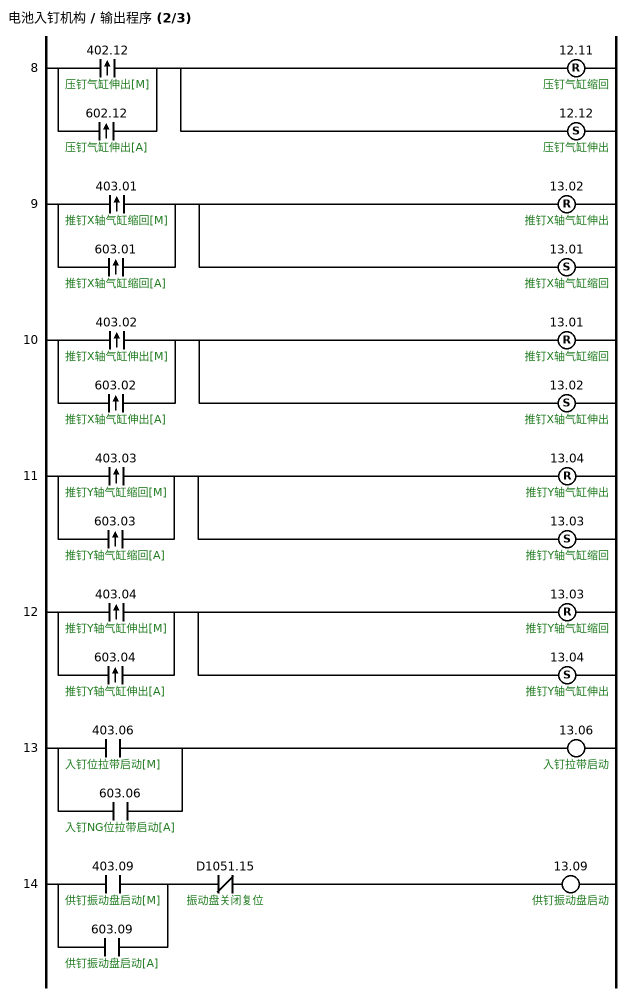
; [picture p120: 电池入钉机构 / 输出程序, rungs 8-14]
; rung 8
@LD 402.12  ; 压钉气缸伸出[M]
@OR 602.12  ; 压钉气缸伸出[A]
RSET 12.11  ; 压钉气缸缩回
SET 12.12  ; 压钉气缸伸出
; rung 9
@LD 403.01  ; 推钉X轴气缸缩回[M]
@OR 603.01  ; 推钉X轴气缸缩回[A]
RSET 13.02  ; 推钉X轴气缸伸出
SET 13.01  ; 推钉X轴气缸缩回
; rung 10
@LD 403.02  ; 推钉X轴气缸伸出[M]
@OR 603.02  ; 推钉X轴气缸伸出[A]
RSET 13.01  ; 推钉X轴气缸缩回
SET 13.02  ; 推钉X轴气缸伸出
; rung 11
@LD 403.03  ; 推钉Y轴气缸缩回[M]
@OR 603.03  ; 推钉Y轴气缸缩回[A]
RSET 13.04  ; 推钉Y轴气缸伸出
SET 13.03  ; 推钉Y轴气缸缩回
; rung 12
@LD 403.04  ; 推钉Y轴气缸伸出[M]
@OR 603.04  ; 推钉Y轴气缸伸出[A]
RSET 13.03  ; 推钉Y轴气缸缩回
SET 13.04  ; 推钉Y轴气缸伸出
; rung 13
LD 403.06  ; 入钉位拉带启动[M]
OR 603.06  ; 入钉NG位拉带启动[A]
OUT 13.06  ; 入钉拉带启动
; rung 14
LD 403.09  ; 供钉振动盘启动[M]
OR 603.09  ; 供钉振动盘启动[A]
ANDNOT D1051.15  ; 振动盘关闭复位
OUT 13.09  ; 供钉振动盘启动

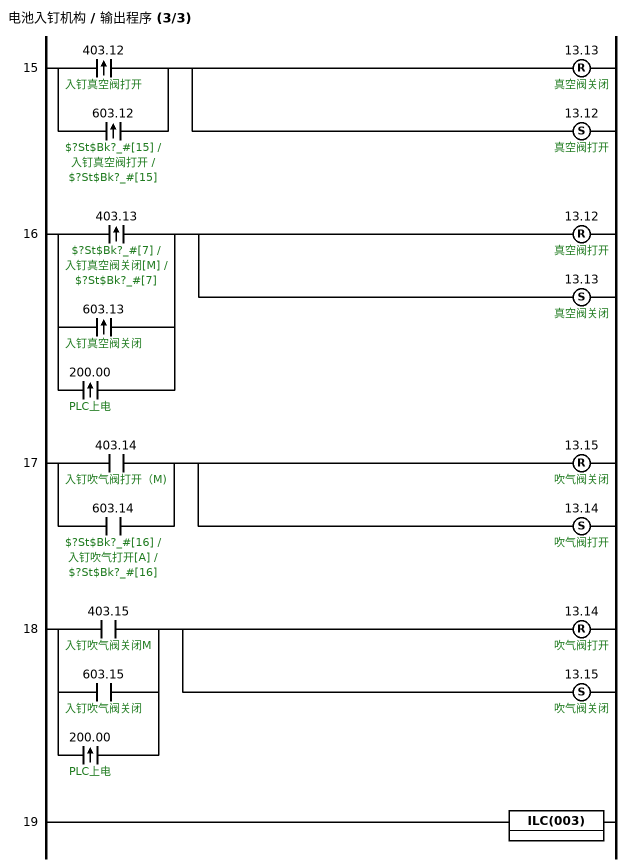
; rung 15
@LD 403.12  ; 入钉真空阀打开
@OR 603.12  ; $?St$Bk?_#[15] / 入钉真空阀打开 / $?St$Bk?_#[15]
RSET 13.13  ; 真空阀关闭
SET 13.12  ; 真空阀打开
; rung 16
@LD 403.13  ; $?St$Bk?_#[7] / 入钉真空阀关闭[M] / $?St$Bk?_#[7]
@OR 603.13  ; 入钉真空阀关闭
@OR 200.00  ; PLC上电
RSET 13.12  ; 真空阀打开
SET 13.13  ; 真空阀关闭
; rung 17
LD 403.14  ; 入钉吹气阀打开（M)
OR 603.14  ; $?St$Bk?_#[16] / 入钉吹气打开[A] / $?St$Bk?_#[16]
RSET 13.15  ; 吹气阀关闭
SET 13.14  ; 吹气阀打开
; rung 18
LD 403.15  ; 入钉吹气阀关闭M
OR 603.15  ; 入钉吹气阀关闭
@OR 200.00  ; PLC上电
RSET 13.14  ; 吹气阀打开
SET 13.15  ; 吹气阀关闭
; rung 19
ILC(003)

### Section 入钉升降伺服参数

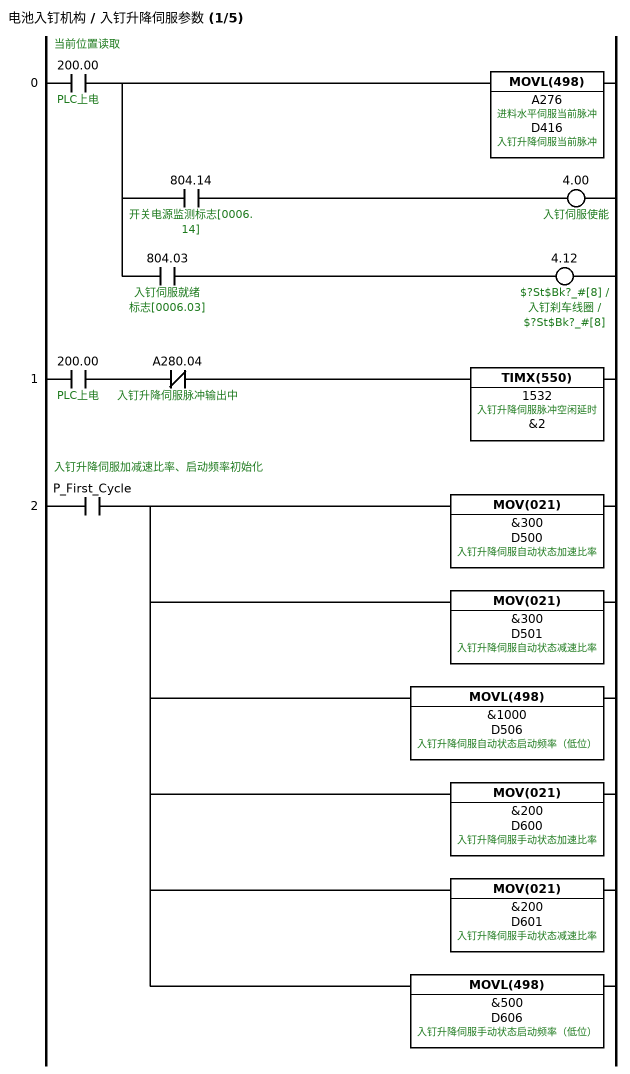
; rung 0: 当前位置读取
LD 200.00  ; PLC上电
OUT TR0
MOVL(498) A276 D416  ; 进料水平伺服当前脉冲, 入钉升降伺服当前脉冲
AND 804.14  ; 开关电源监测标志[0006.14]
OUT 4.00  ; 入钉伺服使能
LD TR0
AND 804.03  ; 入钉伺服就绪 标志[0006.03]
OUT 4.12  ; $?St$Bk?_#[8] / 入钉刹车线圈 / $?St$Bk?_#[8]
; rung 1
LD 200.00  ; PLC上电
ANDNOT A280.04  ; 入钉升降伺服脉冲输出中
TIMX(550) 1532 &2  ; 入钉升降伺服脉冲空闲延时
; rung 2: 入钉升降伺服加减速比率、启动频率初始化
LD P_First_Cycle
MOV(021) &300 D500  ; 入钉升降伺服自动状态加速比率
MOV(021) &300 D501  ; 入钉升降伺服自动状态减速比率
MOVL(498) &1000 D506  ; 入钉升降伺服自动状态启动频率（低位）
MOV(021) &200 D600  ; 入钉升降伺服手动状态加速比率
MOV(021) &200 D601  ; 入钉升降伺服手动状态减速比率
MOVL(498) &500 D606  ; 入钉升降伺服手动状态启动频率（低位）

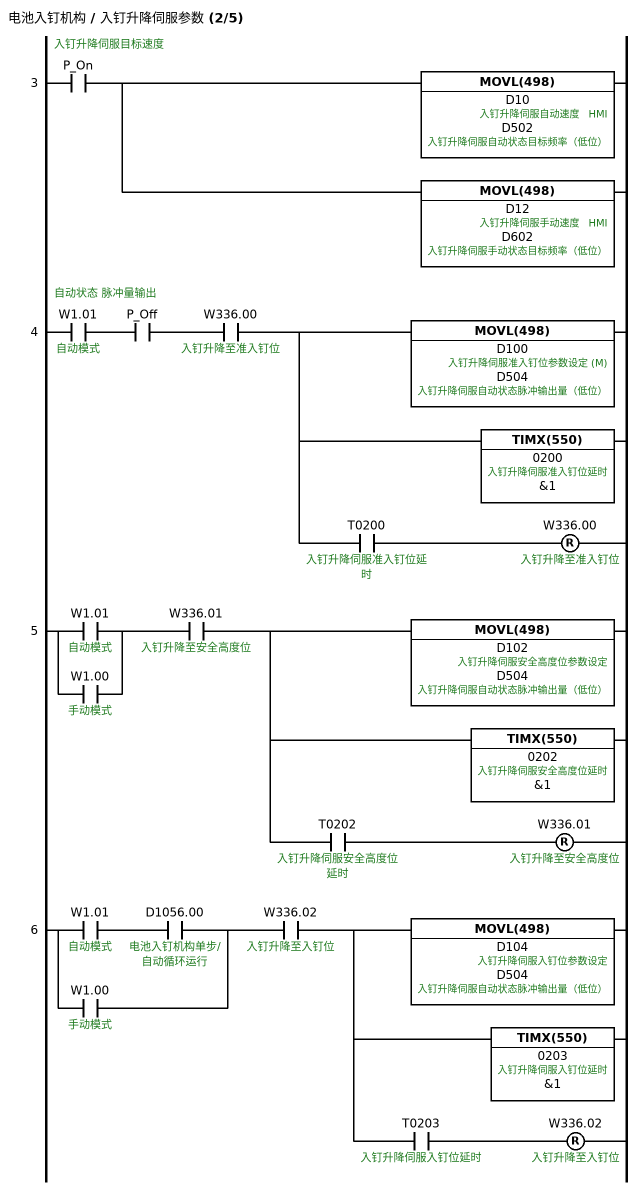
; rung 3: 入钉升降伺服目标速度
LD P_On
MOVL(498) D10 D502  ; 入钉升降伺服自动速度   HMI, 入钉升降伺服自动状态目标频率（低位）
MOVL(498) D12 D602  ; 入钉升降伺服手动速度   HMI, 入钉升降伺服手动状态目标频率（低位）
; rung 4: 自动状态 脉冲量输出
LD W1.01  ; 自动模式
AND P_Off
AND W336.00  ; 入钉升降至准入钉位
MOVL(498) D100 D504  ; 入钉升降伺服准入钉位参数设定 (M), 入钉升降伺服自动状态脉冲输出量（低位）
TIMX(550) 0200 &1  ; 入钉升降伺服准入钉位延时
AND T0200  ; 入钉升降伺服准入钉位延时
RSET W336.00  ; 入钉升降至准入钉位
; rung 5
LD W1.01  ; 自动模式
OR W1.00  ; 手动模式
AND W336.01  ; 入钉升降至安全高度位
MOVL(498) D102 D504  ; 入钉升降伺服安全高度位参数设定, 入钉升降伺服自动状态脉冲输出量（低位）
TIMX(550) 0202 &1  ; 入钉升降伺服安全高度位延时
AND T0202  ; 入钉升降伺服安全高度位延时
RSET W336.01  ; 入钉升降至安全高度位
; rung 6
LD W1.01  ; 自动模式
AND D1056.00  ; 电池入钉机构单步/自动循环运行
OR W1.00  ; 手动模式
AND W336.02  ; 入钉升降至入钉位
MOVL(498) D104 D504  ; 入钉升降伺服入钉位参数设定, 入钉升降伺服自动状态脉冲输出量（低位）
TIMX(550) 0203 &1  ; 入钉升降伺服入钉位延时
AND T0203  ; 入钉升降伺服入钉位延时
RSET W336.02  ; 入钉升降至入钉位

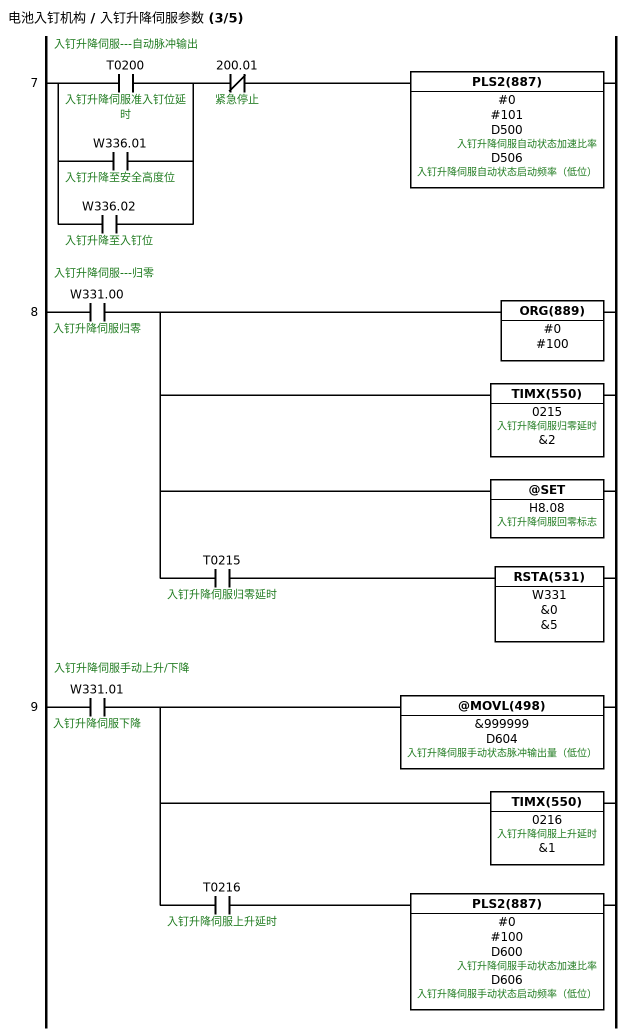
; rung 7: 入钉升降伺服---自动脉冲输出
LD T0200  ; 入钉升降伺服准入钉位延时
OR W336.01  ; 入钉升降至安全高度位
OR W336.02  ; 入钉升降至入钉位
ANDNOT 200.01  ; 紧急停止
PLS2(887) #0 #101 D500 D506  ; 入钉升降伺服自动状态加速比率, 入钉升降伺服自动状态启动频率（低位）
; rung 8: 入钉升降伺服---归零
LD W331.00  ; 入钉升降伺服归零
ORG(889) #0 #100
TIMX(550) 0215 &2  ; 入钉升降伺服归零延时
@SET H8.08  ; 入钉升降伺服回零标志
AND T0215  ; 入钉升降伺服归零延时
RSTA(531) W331 &0 &5
; rung 9: 入钉升降伺服手动上升/下降
LD W331.01  ; 入钉升降伺服下降
@MOVL(498) &999999 D604  ; 入钉升降伺服手动状态脉冲输出量（低位）
TIMX(550) 0216 &1  ; 入钉升降伺服上升延时
AND T0216  ; 入钉升降伺服上升延时
PLS2(887) #0 #100 D600 D606  ; 入钉升降伺服手动状态加速比率, 入钉升降伺服手动状态启动频率（低位）

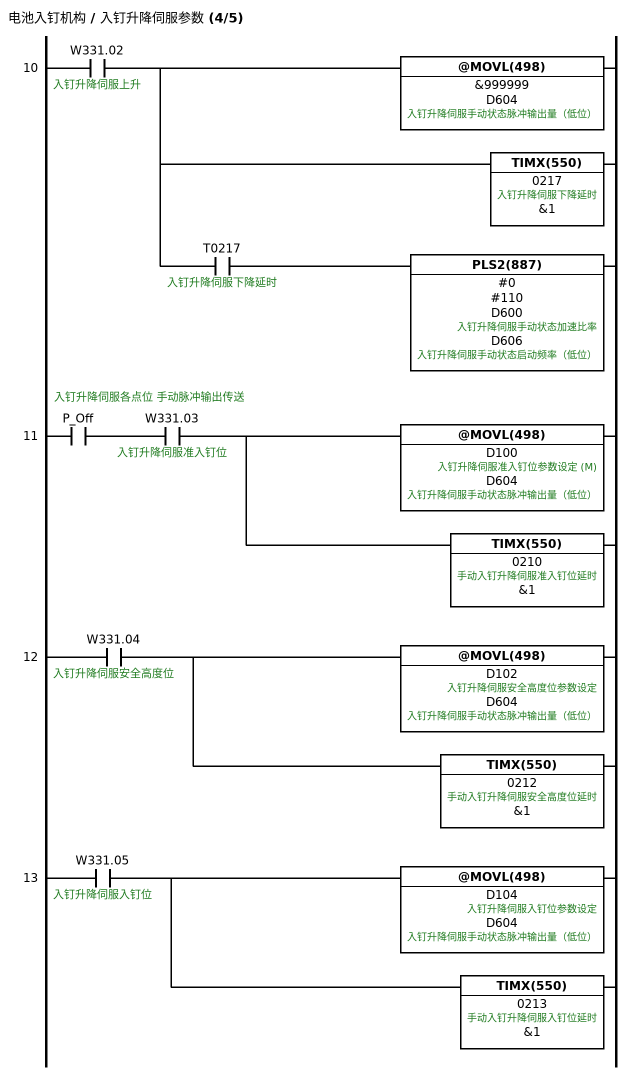
; rung 10
LD W331.02  ; 入钉升降伺服上升
@MOVL(498) &999999 D604  ; 入钉升降伺服手动状态脉冲输出量（低位）
TIMX(550) 0217 &1  ; 入钉升降伺服下降延时
AND T0217  ; 入钉升降伺服下降延时
PLS2(887) #0 #110 D600 D606  ; 入钉升降伺服手动状态加速比率, 入钉升降伺服手动状态启动频率（低位）
; rung 11: 入钉升降伺服各点位 手动脉冲输出传送
LD P_Off
AND W331.03  ; 入钉升降伺服准入钉位
@MOVL(498) D100 D604  ; 入钉升降伺服准入钉位参数设定 (M), 入钉升降伺服手动状态脉冲输出量（低位）
TIMX(550) 0210 &1  ; 手动入钉升降伺服准入钉位延时
; rung 12
LD W331.04  ; 入钉升降伺服安全高度位
@MOVL(498) D102 D604  ; 入钉升降伺服安全高度位参数设定, 入钉升降伺服手动状态脉冲输出量（低位）
TIMX(550) 0212 &1  ; 手动入钉升降伺服安全高度位延时
; rung 13
LD W331.05  ; 入钉升降伺服入钉位
@MOVL(498) D104 D604  ; 入钉升降伺服入钉位参数设定, 入钉升降伺服手动状态脉冲输出量（低位）
TIMX(550) 0213 &1  ; 手动入钉升降伺服入钉位延时

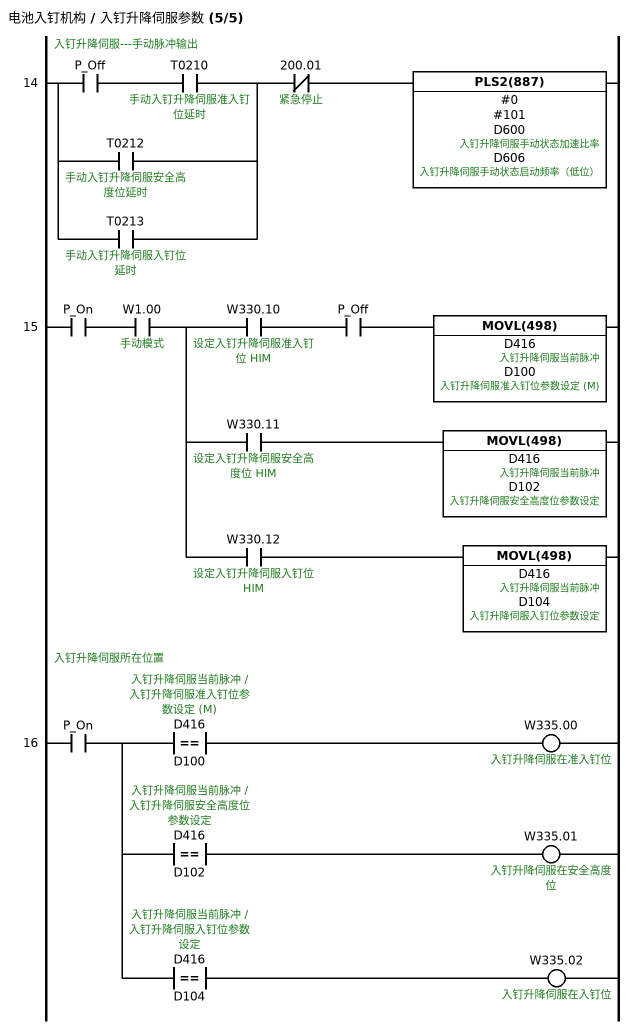
; rung 14: 入钉升降伺服---手动脉冲输出
LD P_Off
AND T0210  ; 手动入钉升降伺服准入钉位延时
OR T0212  ; 手动入钉升降伺服安全高度位延时
OR T0213  ; 手动入钉升降伺服入钉位延时
ANDNOT 200.01  ; 紧急停止
PLS2(887) #0 #101 D600 D606  ; 入钉升降伺服手动状态加速比率, 入钉升降伺服手动状态启动频率（低位）
; rung 15
LD P_On
AND W1.00  ; 手动模式
OUT TR0
AND W330.10  ; 设定入钉升降伺服准入钉位 HIM
AND P_Off
MOVL(498) D416 D100  ; 入钉升降伺服当前脉冲, 入钉升降伺服准入钉位参数设定 (M)
LD TR0
AND W330.11  ; 设定入钉升降伺服安全高度位 HIM
MOVL(498) D416 D102  ; 入钉升降伺服当前脉冲, 入钉升降伺服安全高度位参数设定
LD TR0
AND W330.12  ; 设定入钉升降伺服入钉位 HIM
MOVL(498) D416 D104  ; 入钉升降伺服当前脉冲, 入钉升降伺服入钉位参数设定
; rung 16: 入钉升降伺服所在位置
LD P_On
OUT TR0
AND=SL(303) D416 D100  ; 入钉升降伺服当前脉冲, 入钉升降伺服准入钉位参数设定 (M)
OUT W335.00  ; 入钉升降伺服在准入钉位
LD TR0
AND=SL(303) D416 D102  ; 入钉升降伺服当前脉冲, 入钉升降伺服安全高度位参数设定
OUT W335.01  ; 入钉升降伺服在安全高度位
LD TR0
AND=SL(303) D416 D104  ; 入钉升降伺服当前脉冲, 入钉升降伺服入钉位参数设定
OUT W335.02  ; 入钉升降伺服在入钉位

### Section 入钉旋转步进参数

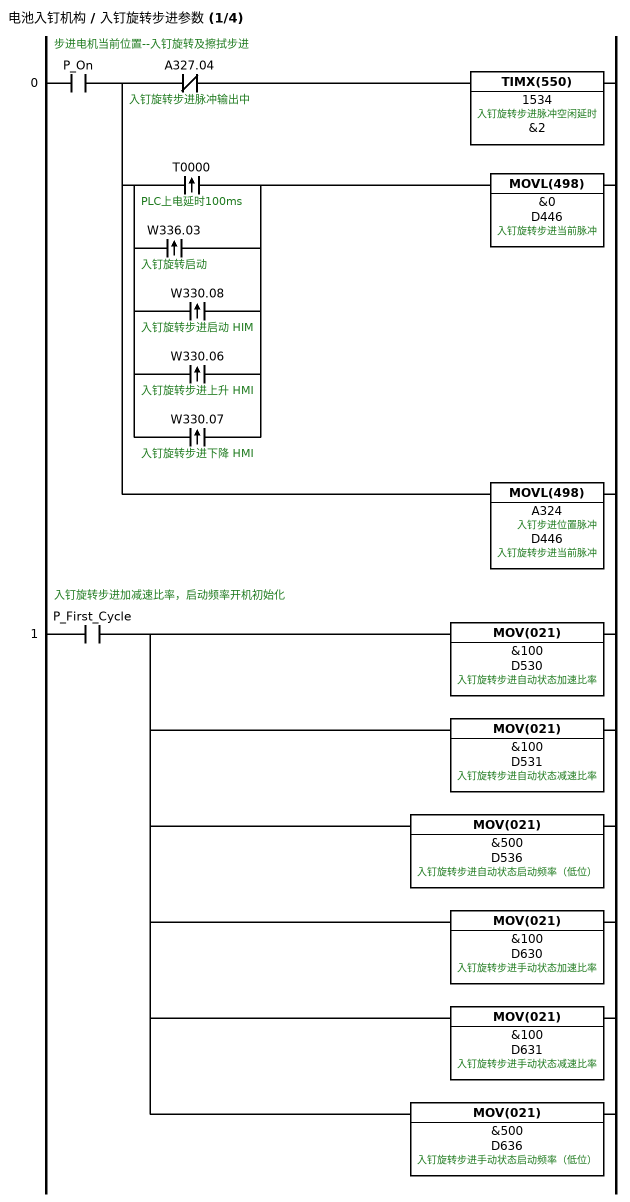
; rung 0: 步进电机当前位置--入钉旋转及擦拭步进
LD P_On
OUT TR0
ANDNOT A327.04  ; 入钉旋转步进脉冲输出中
TIMX(550) 1534 &2  ; 入钉旋转步进脉冲空闲延时
LD TR0
@LD T0000  ; PLC上电延时100ms
@OR W336.03  ; 入钉旋转启动
@OR W330.08  ; 入钉旋转步进启动 HIM
@OR W330.06  ; 入钉旋转步进上升 HMI
@OR W330.07  ; 入钉旋转步进下降 HMI
ANDLD
MOVL(498) &0 D446  ; 入钉旋转步进当前脉冲
LD TR0
MOVL(498) A324 D446  ; 入钉步进位置脉冲, 入钉旋转步进当前脉冲
; rung 1: 入钉旋转步进加减速比率，启动频率开机初始化
LD P_First_Cycle
MOV(021) &100 D530  ; 入钉旋转步进自动状态加速比率
MOV(021) &100 D531  ; 入钉旋转步进自动状态减速比率
MOV(021) &500 D536  ; 入钉旋转步进自动状态启动频率（低位）
MOV(021) &100 D630  ; 入钉旋转步进手动状态加速比率
MOV(021) &100 D631  ; 入钉旋转步进手动状态减速比率
MOV(021) &500 D636  ; 入钉旋转步进手动状态启动频率（低位）

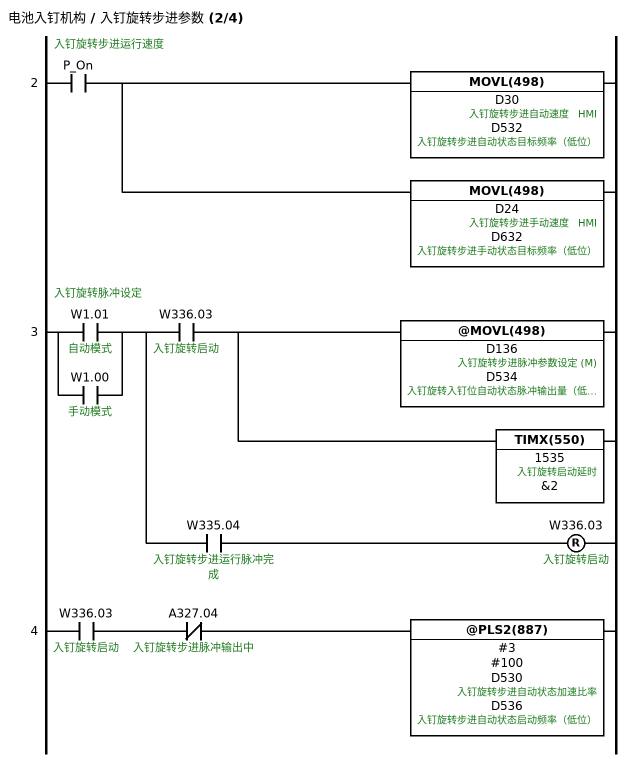
; rung 2: 入钉旋转步进运行速度
LD P_On
MOVL(498) D30 D532  ; 入钉旋转步进自动速度   HMI, 入钉旋转步进自动状态目标频率（低位）
MOVL(498) D24 D632  ; 入钉旋转步进手动速度   HMI, 入钉旋转步进手动状态目标频率（低位）
; rung 3: 入钉旋转脉冲设定
LD W1.01  ; 自动模式
OR W1.00  ; 手动模式
OUT TR0
AND W336.03  ; 入钉旋转启动
@MOVL(498) D136 D534  ; 入钉旋转步进脉冲参数设定 (M), 入钉旋转入钉位自动状态脉冲输出量（低位）
TIMX(550) 1535 &2  ; 入钉旋转启动延时
LD TR0
AND W335.04  ; 入钉旋转步进运行脉冲完成
RSET W336.03  ; 入钉旋转启动
; rung 4
LD W336.03  ; 入钉旋转启动
ANDNOT A327.04  ; 入钉旋转步进脉冲输出中
@PLS2(887) #3 #100 D530 D536  ; 入钉旋转步进自动状态加速比率, 入钉旋转步进自动状态启动频率（低位）

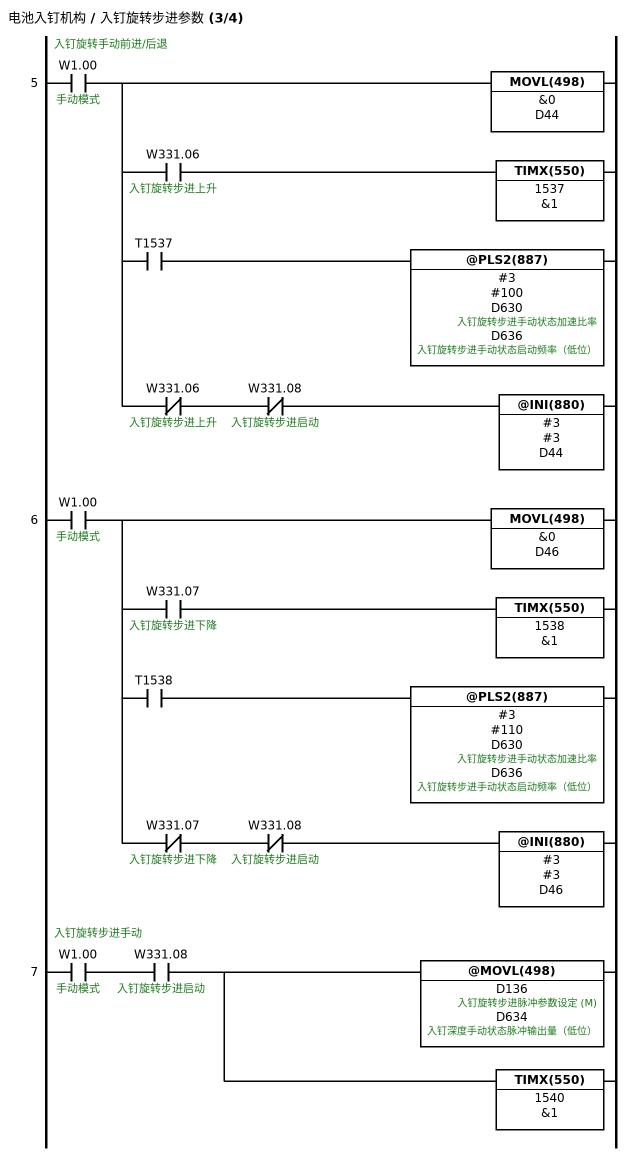
; rung 5: 入钉旋转手动前进/后退
LD W1.00  ; 手动模式
OUT TR0
MOVL(498) &0 D44
AND W331.06  ; 入钉旋转步进上升
TIMX(550) 1537 &1
LD TR0
AND T1537
@PLS2(887) #3 #100 D630 D636  ; 入钉旋转步进手动状态加速比率, 入钉旋转步进手动状态启动频率（低位）
LD TR0
ANDNOT W331.06  ; 入钉旋转步进上升
ANDNOT W331.08  ; 入钉旋转步进启动
@INI(880) #3 #3 D44
; rung 6
LD W1.00  ; 手动模式
OUT TR0
MOVL(498) &0 D46
AND W331.07  ; 入钉旋转步进下降
TIMX(550) 1538 &1
LD TR0
AND T1538
@PLS2(887) #3 #110 D630 D636  ; 入钉旋转步进手动状态加速比率, 入钉旋转步进手动状态启动频率（低位）
LD TR0
ANDNOT W331.07  ; 入钉旋转步进下降
ANDNOT W331.08  ; 入钉旋转步进启动
@INI(880) #3 #3 D46
; rung 7: 入钉旋转步进手动
LD W1.00  ; 手动模式
AND W331.08  ; 入钉旋转步进启动
@MOVL(498) D136 D634  ; 入钉旋转步进脉冲参数设定 (M), 入钉深度手动状态脉冲输出量（低位）
TIMX(550) 1540 &1

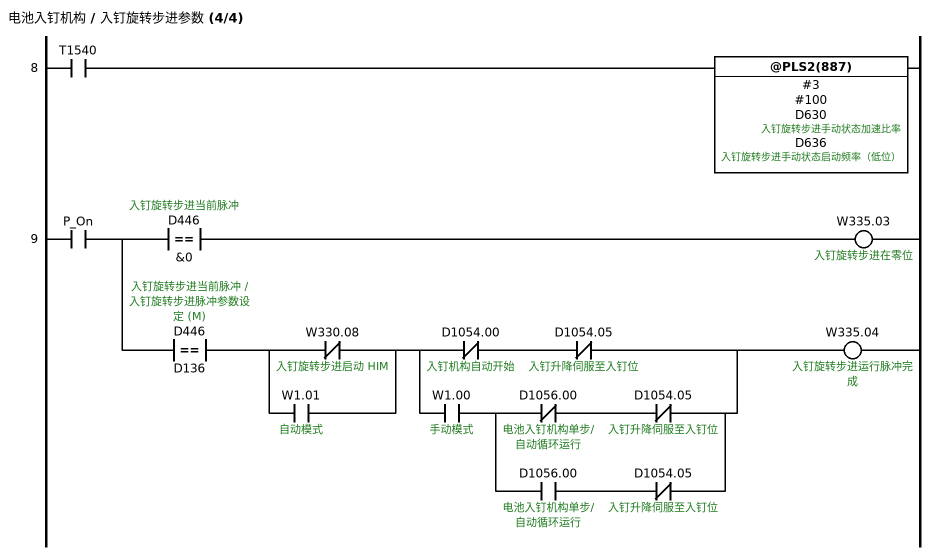
; rung 8
LD T1540
@PLS2(887) #3 #100 D630 D636  ; 入钉旋转步进手动状态加速比率, 入钉旋转步进手动状态启动频率（低位）
; rung 9
LD P_On
OUT TR0
AND=SL(303) D446 &0  ; 入钉旋转步进当前脉冲
OUT W335.03  ; 入钉旋转步进在零位
LD TR0
AND=SL(303) D446 D136  ; 入钉旋转步进当前脉冲, 入钉旋转步进脉冲参数设定 (M)
LDNOT W330.08  ; 入钉旋转步进启动 HIM
OR W1.01  ; 自动模式
ANDLD
LDNOT D1054.00  ; 入钉机构自动开始
ANDNOT D1054.05  ; 入钉升降伺服至入钉位
LD W1.00  ; 手动模式
LDNOT D1056.00  ; 电池入钉机构单步/自动循环运行
ANDNOT D1054.05  ; 入钉升降伺服至入钉位
LD D1056.00  ; 电池入钉机构单步/自动循环运行
ANDNOT D1054.05  ; 入钉升降伺服至入钉位
ORLD
ANDLD
ORLD
ANDLD
OUT W335.04  ; 入钉旋转步进运行脉冲完成

### Section END
; rung 0
END(001)

## Program 入钉NG抓取机构 (cyclic task 5)

### Section 主程序

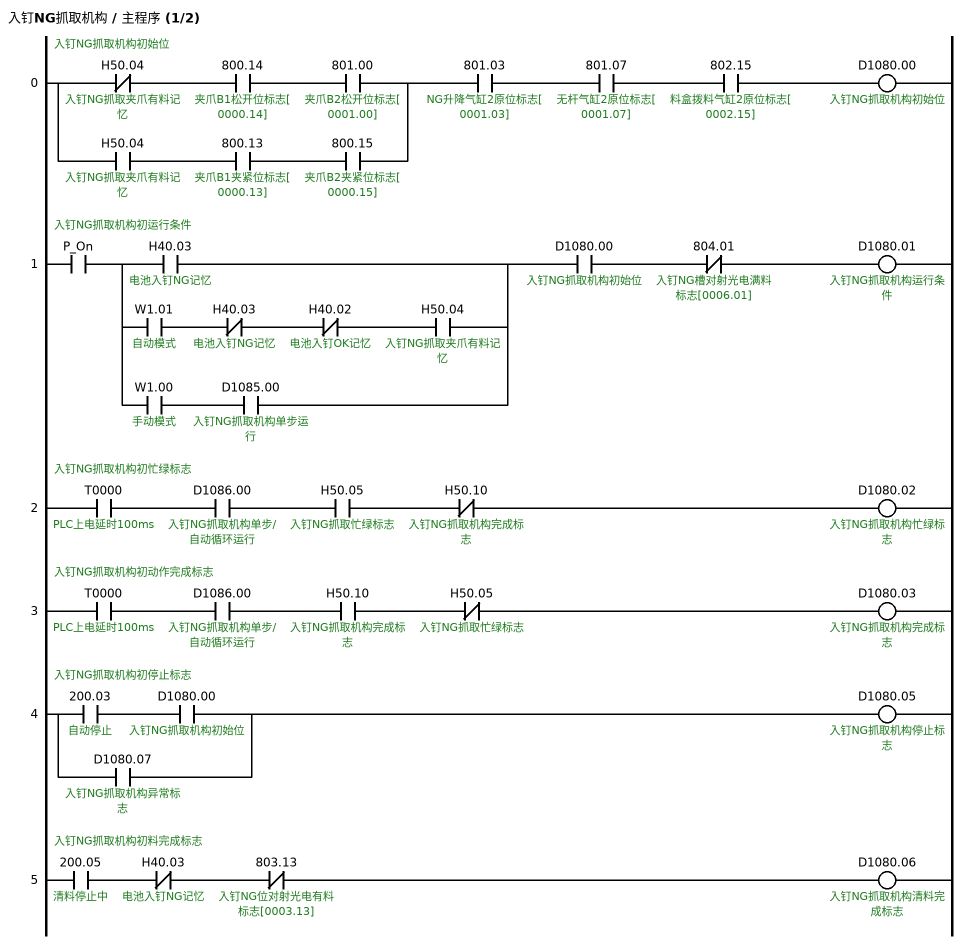
; rung 0: 入钉NG抓取机构初始位
LDNOT H50.04  ; 入钉NG抓取夹爪有料记忆
AND 800.14  ; 夹爪B1松开位标志[0000.14]
AND 801.00  ; 夹爪B2松开位标志[0001.00]
LD H50.04  ; 入钉NG抓取夹爪有料记忆
AND 800.13  ; 夹爪B1夹紧位标志[0000.13]
AND 800.15  ; 夹爪B2夹紧位标志[0000.15]
ORLD
AND 801.03  ; NG升降气缸2原位标志[0001.03]
AND 801.07  ; 无杆气缸2原位标志[0001.07]
AND 802.15  ; 料盒拨料气缸2原位标志[0002.15]
OUT D1080.00  ; 入钉NG抓取机构初始位
; rung 1: 入钉NG抓取机构初运行条件
LD P_On
LD H40.03  ; 电池入钉NG记忆
LD W1.01  ; 自动模式
ANDNOT H40.03  ; 电池入钉NG记忆
ANDNOT H40.02  ; 电池入钉OK记忆
AND H50.04  ; 入钉NG抓取夹爪有料记忆
ORLD
LD W1.00  ; 手动模式
AND D1085.00  ; 入钉NG抓取机构单步运行
ORLD
ANDLD
AND D1080.00  ; 入钉NG抓取机构初始位
ANDNOT 804.01  ; 入钉NG槽对射光电满料标志[0006.01]
OUT D1080.01  ; 入钉NG抓取机构运行条件
; rung 2: 入钉NG抓取机构初忙绿标志
LD T0000  ; PLC上电延时100ms
AND D1086.00  ; 入钉NG抓取机构单步/自动循环运行
AND H50.05  ; 入钉NG抓取忙绿标志
ANDNOT H50.10  ; 入钉NG抓取机构完成标志
OUT D1080.02  ; 入钉NG抓取机构忙绿标志
; rung 3: 入钉NG抓取机构初动作完成标志
LD T0000  ; PLC上电延时100ms
AND D1086.00  ; 入钉NG抓取机构单步/自动循环运行
AND H50.10  ; 入钉NG抓取机构完成标志
ANDNOT H50.05  ; 入钉NG抓取忙绿标志
OUT D1080.03  ; 入钉NG抓取机构完成标志
; rung 4: 入钉NG抓取机构初停止标志
LD 200.03  ; 自动停止
AND D1080.00  ; 入钉NG抓取机构初始位
OR D1080.07  ; 入钉NG抓取机构异常标志
OUT D1080.05  ; 入钉NG抓取机构停止标志
; rung 5: 入钉NG抓取机构初料完成标志
LD 200.05  ; 清料停止中
ANDNOT H40.03  ; 电池入钉NG记忆
ANDNOT 803.13  ; 入钉NG位对射光电有料标志[0003.13]
OUT D1080.06  ; 入钉NG抓取机构清料完成标志

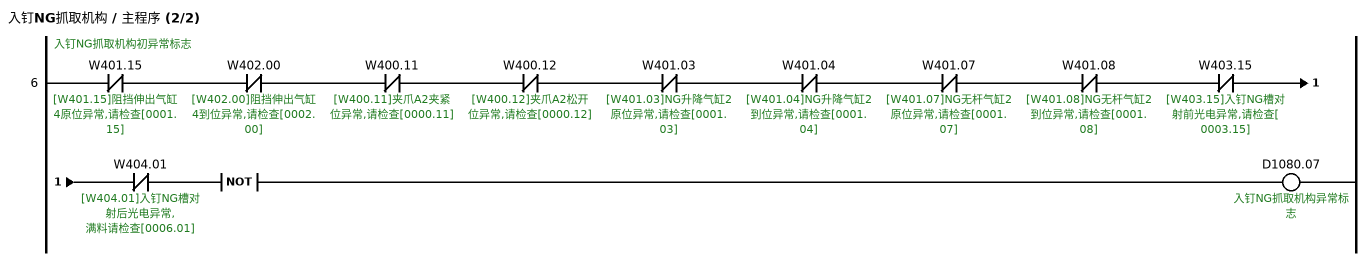
; rung 6: 入钉NG抓取机构初异常标志
LDNOT W401.15  ; [W401.15]阻挡伸出气缸4原位异常,请检查[0001.15]
ANDNOT W402.00  ; [W402.00]阻挡伸出气缸4到位异常,请检查[0002.00]
ANDNOT W400.11  ; [W400.11]夹爪A2夹紧位异常,请检查[0000.11]
ANDNOT W400.12  ; [W400.12]夹爪A2松开位异常,请检查[0000.12]
ANDNOT W401.03  ; [W401.03]NG升降气缸2原位异常,请检查[0001.03]
ANDNOT W401.04  ; [W401.04]NG升降气缸2到位异常,请检查[0001.04]
ANDNOT W401.07  ; [W401.07]NG无杆气缸2原位异常,请检查[0001.07]
ANDNOT W401.08  ; [W401.08]NG无杆气缸2到位异常,请检查[0001.08]
ANDNOT W403.15  ; [W403.15]入钉NG槽对射前光电异常,请检查[0003.15]
ANDNOT W404.01  ; [W404.01]入钉NG槽对射后光电异常,满料请检查[0006.01]
NOT(520)
OUT D1080.07  ; 入钉NG抓取机构异常标志

### Section 工站复位

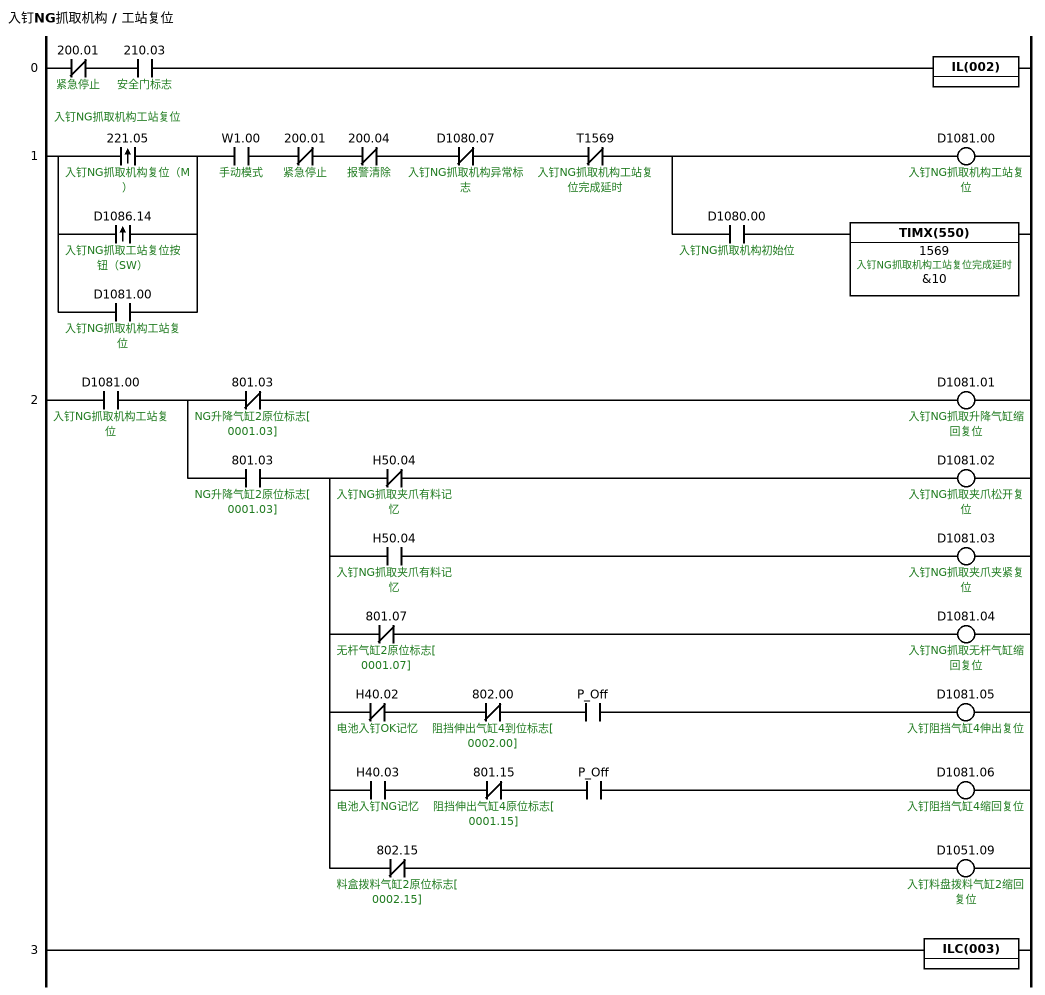
; rung 0
LDNOT 200.01  ; 紧急停止
AND 210.03  ; 安全门标志
IL(002)
; rung 1: 入钉NG抓取机构工站复位
@LD 221.05  ; 入钉NG抓取机构复位（M）
@OR D1086.14  ; 入钉NG抓取工站复位按钮（SW）
OR D1081.00  ; 入钉NG抓取机构工站复位
AND W1.00  ; 手动模式
ANDNOT 200.01  ; 紧急停止
ANDNOT 200.04  ; 报警清除
ANDNOT D1080.07  ; 入钉NG抓取机构异常标志
ANDNOT T1569  ; 入钉NG抓取机构工站复位完成延时
OUT D1081.00  ; 入钉NG抓取机构工站复位
AND D1080.00  ; 入钉NG抓取机构初始位
TIMX(550) 1569 &10  ; 入钉NG抓取机构工站复位完成延时
; rung 2
LD D1081.00  ; 入钉NG抓取机构工站复位
OUT TR0
ANDNOT 801.03  ; NG升降气缸2原位标志[0001.03]
OUT D1081.01  ; 入钉NG抓取升降气缸缩回复位
LD TR0
AND 801.03  ; NG升降气缸2原位标志[0001.03]
OUT TR0
ANDNOT H50.04  ; 入钉NG抓取夹爪有料记忆
OUT D1081.02  ; 入钉NG抓取夹爪松开复位
LD TR0
AND H50.04  ; 入钉NG抓取夹爪有料记忆
OUT D1081.03  ; 入钉NG抓取夹爪夹紧复位
LD TR0
ANDNOT 801.07  ; 无杆气缸2原位标志[0001.07]
OUT D1081.04  ; 入钉NG抓取无杆气缸缩回复位
LD TR0
ANDNOT H40.02  ; 电池入钉OK记忆
ANDNOT 802.00  ; 阻挡伸出气缸4到位标志[0002.00]
AND P_Off
OUT D1081.05  ; 入钉阻挡气缸4伸出复位
LD TR0
AND H40.03  ; 电池入钉NG记忆
ANDNOT 801.15  ; 阻挡伸出气缸4原位标志[0001.15]
AND P_Off
OUT D1081.06  ; 入钉阻挡气缸4缩回复位
LD TR0
ANDNOT 802.15  ; 料盒拨料气缸2原位标志[0002.15]
OUT D1051.09  ; 入钉料盘拨料气缸2缩回复位
; rung 3
ILC(003)

### Section 手动程序

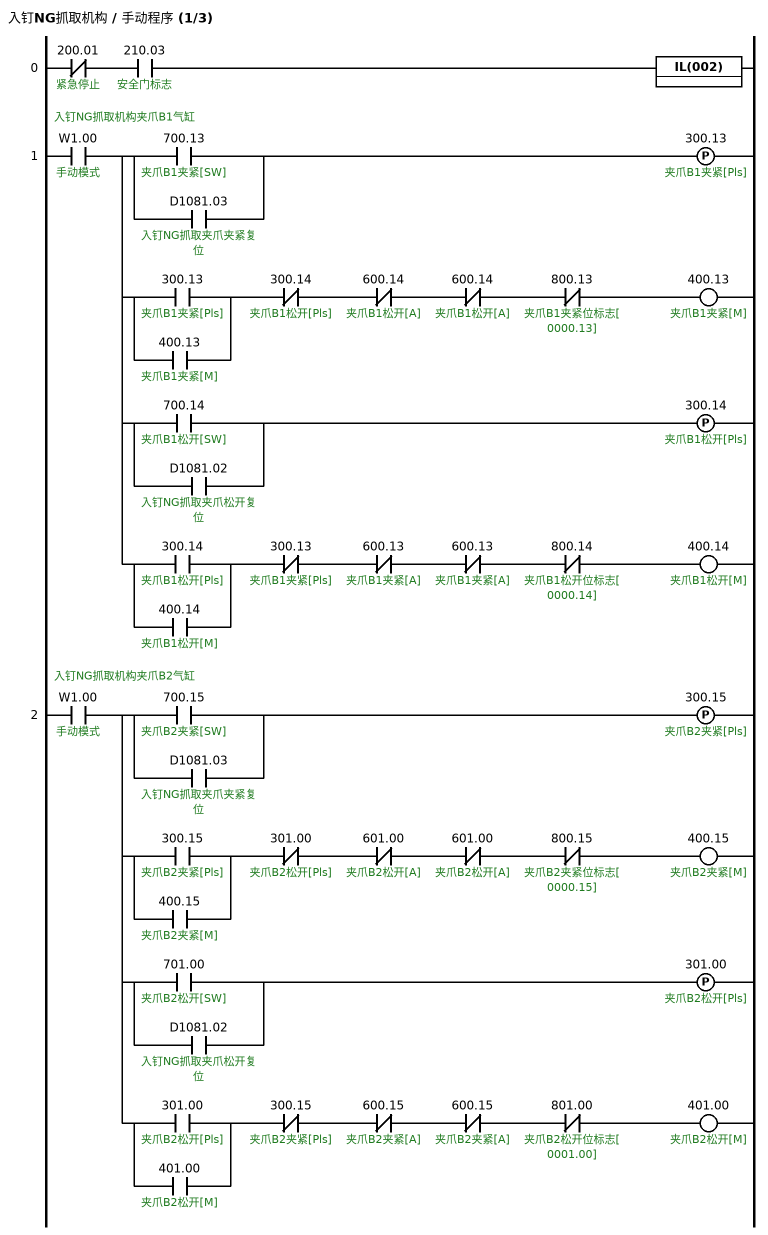
; rung 0
LDNOT 200.01  ; 紧急停止
AND 210.03  ; 安全门标志
IL(002)
; rung 1: 入钉NG抓取机构夹爪B1气缸
LD W1.00  ; 手动模式
OUT TR0
LD 700.13  ; 夹爪B1夹紧[SW]
OR D1081.03  ; 入钉NG抓取夹爪夹紧复位
ANDLD
DIFU(013) 300.13  ; 夹爪B1夹紧[Pls]
LD TR0
LD 300.13  ; 夹爪B1夹紧[Pls]
OR 400.13  ; 夹爪B1夹紧[M]
ANDLD
ANDNOT 300.14  ; 夹爪B1松开[Pls]
ANDNOT 600.14  ; 夹爪B1松开[A]
ANDNOT 600.14  ; 夹爪B1松开[A]
ANDNOT 800.13  ; 夹爪B1夹紧位标志[0000.13]
OUT 400.13  ; 夹爪B1夹紧[M]
LD TR0
LD 700.14  ; 夹爪B1松开[SW]
OR D1081.02  ; 入钉NG抓取夹爪松开复位
ANDLD
DIFU(013) 300.14  ; 夹爪B1松开[Pls]
LD TR0
LD 300.14  ; 夹爪B1松开[Pls]
OR 400.14  ; 夹爪B1松开[M]
ANDLD
ANDNOT 300.13  ; 夹爪B1夹紧[Pls]
ANDNOT 600.13  ; 夹爪B1夹紧[A]
ANDNOT 600.13  ; 夹爪B1夹紧[A]
ANDNOT 800.14  ; 夹爪B1松开位标志[0000.14]
OUT 400.14  ; 夹爪B1松开[M]
; rung 2: 入钉NG抓取机构夹爪B2气缸
LD W1.00  ; 手动模式
OUT TR0
LD 700.15  ; 夹爪B2夹紧[SW]
OR D1081.03  ; 入钉NG抓取夹爪夹紧复位
ANDLD
DIFU(013) 300.15  ; 夹爪B2夹紧[Pls]
LD TR0
LD 300.15  ; 夹爪B2夹紧[Pls]
OR 400.15  ; 夹爪B2夹紧[M]
ANDLD
ANDNOT 301.00  ; 夹爪B2松开[Pls]
ANDNOT 601.00  ; 夹爪B2松开[A]
ANDNOT 601.00  ; 夹爪B2松开[A]
ANDNOT 800.15  ; 夹爪B2夹紧位标志[0000.15]
OUT 400.15  ; 夹爪B2夹紧[M]
LD TR0
LD 701.00  ; 夹爪B2松开[SW]
OR D1081.02  ; 入钉NG抓取夹爪松开复位
ANDLD
DIFU(013) 301.00  ; 夹爪B2松开[Pls]
LD TR0
LD 301.00  ; 夹爪B2松开[Pls]
OR 401.00  ; 夹爪B2松开[M]
ANDLD
ANDNOT 300.15  ; 夹爪B2夹紧[Pls]
ANDNOT 600.15  ; 夹爪B2夹紧[A]
ANDNOT 600.15  ; 夹爪B2夹紧[A]
ANDNOT 801.00  ; 夹爪B2松开位标志[0001.00]
OUT 401.00  ; 夹爪B2松开[M]

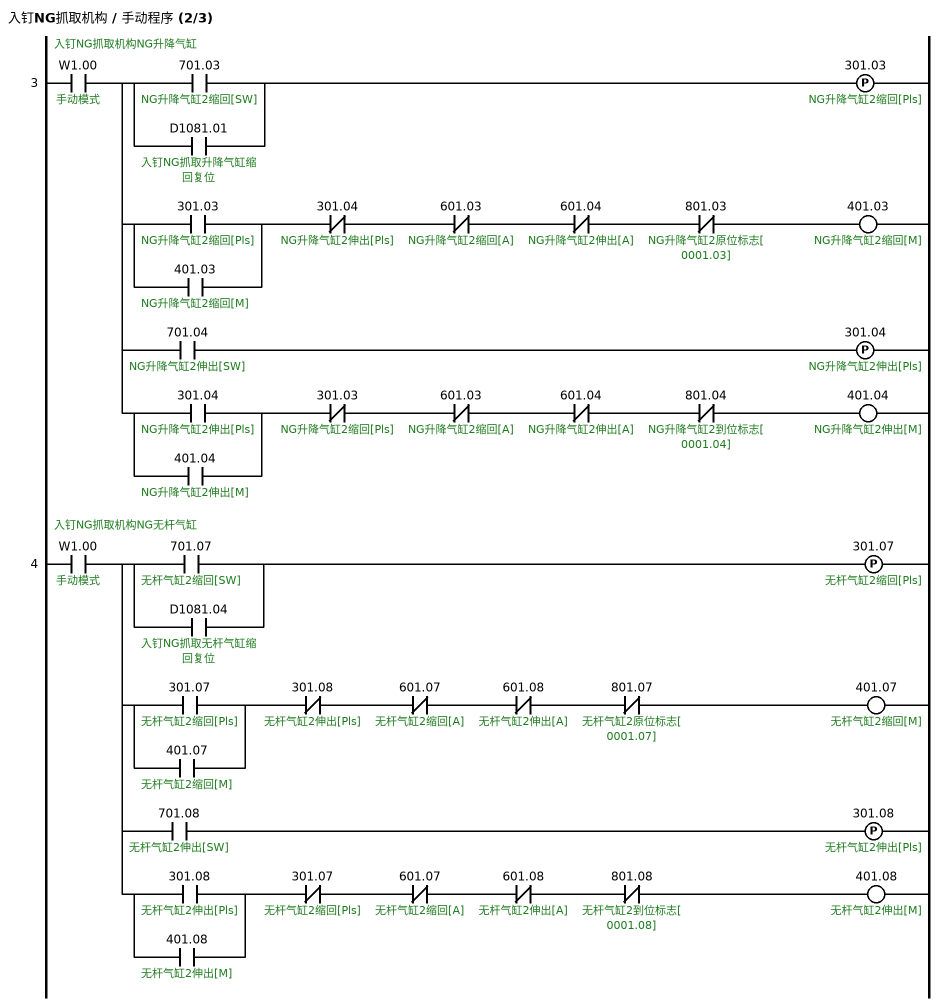
; rung 3: 入钉NG抓取机构NG升降气缸
LD W1.00  ; 手动模式
OUT TR0
LD 701.03  ; NG升降气缸2缩回[SW]
OR D1081.01  ; 入钉NG抓取升降气缸缩回复位
ANDLD
DIFU(013) 301.03  ; NG升降气缸2缩回[Pls]
LD TR0
LD 301.03  ; NG升降气缸2缩回[Pls]
OR 401.03  ; NG升降气缸2缩回[M]
ANDLD
ANDNOT 301.04  ; NG升降气缸2伸出[Pls]
ANDNOT 601.03  ; NG升降气缸2缩回[A]
ANDNOT 601.04  ; NG升降气缸2伸出[A]
ANDNOT 801.03  ; NG升降气缸2原位标志[0001.03]
OUT 401.03  ; NG升降气缸2缩回[M]
LD TR0
AND 701.04  ; NG升降气缸2伸出[SW]
DIFU(013) 301.04  ; NG升降气缸2伸出[Pls]
LD TR0
LD 301.04  ; NG升降气缸2伸出[Pls]
OR 401.04  ; NG升降气缸2伸出[M]
ANDLD
ANDNOT 301.03  ; NG升降气缸2缩回[Pls]
ANDNOT 601.03  ; NG升降气缸2缩回[A]
ANDNOT 601.04  ; NG升降气缸2伸出[A]
ANDNOT 801.04  ; NG升降气缸2到位标志[0001.04]
OUT 401.04  ; NG升降气缸2伸出[M]
; rung 4: 入钉NG抓取机构NG无杆气缸
LD W1.00  ; 手动模式
OUT TR0
LD 701.07  ; 无杆气缸2缩回[SW]
OR D1081.04  ; 入钉NG抓取无杆气缸缩回复位
ANDLD
DIFU(013) 301.07  ; 无杆气缸2缩回[Pls]
LD TR0
LD 301.07  ; 无杆气缸2缩回[Pls]
OR 401.07  ; 无杆气缸2缩回[M]
ANDLD
ANDNOT 301.08  ; 无杆气缸2伸出[Pls]
ANDNOT 601.07  ; 无杆气缸2缩回[A]
ANDNOT 601.08  ; 无杆气缸2伸出[A]
ANDNOT 801.07  ; 无杆气缸2原位标志[0001.07]
OUT 401.07  ; 无杆气缸2缩回[M]
LD TR0
AND 701.08  ; 无杆气缸2伸出[SW]
DIFU(013) 301.08  ; 无杆气缸2伸出[Pls]
LD TR0
LD 301.08  ; 无杆气缸2伸出[Pls]
OR 401.08  ; 无杆气缸2伸出[M]
ANDLD
ANDNOT 301.07  ; 无杆气缸2缩回[Pls]
ANDNOT 601.07  ; 无杆气缸2缩回[A]
ANDNOT 601.08  ; 无杆气缸2伸出[A]
ANDNOT 801.08  ; 无杆气缸2到位标志[0001.08]
OUT 401.08  ; 无杆气缸2伸出[M]

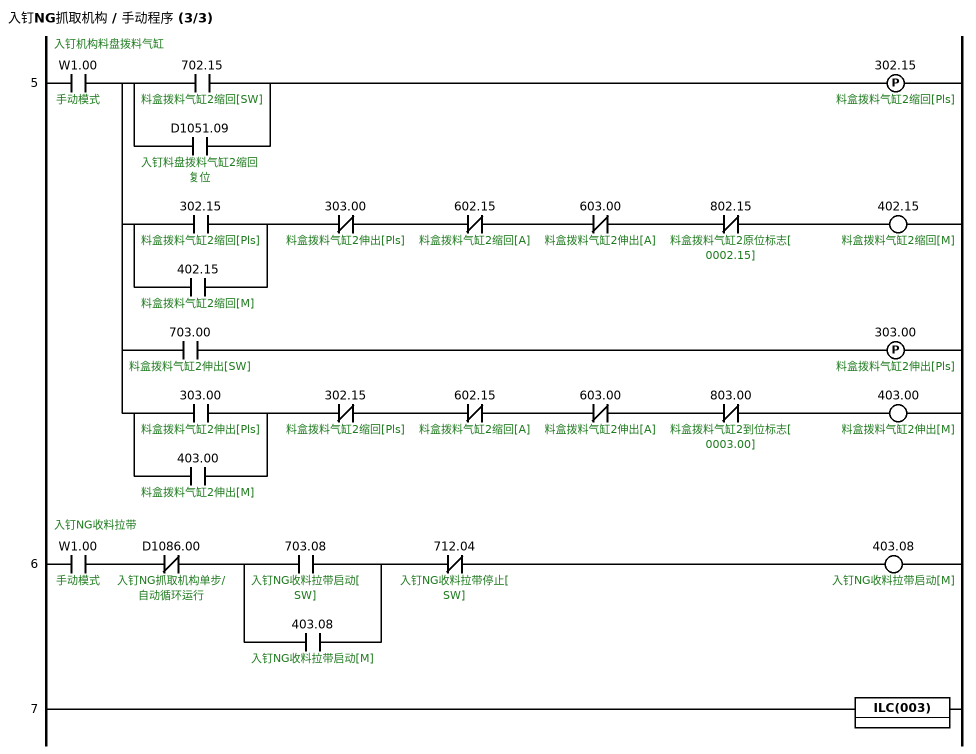
; rung 5: 入钉机构料盘拨料气缸
LD W1.00  ; 手动模式
OUT TR0
LD 702.15  ; 料盒拨料气缸2缩回[SW]
OR D1051.09  ; 入钉料盘拨料气缸2缩回复位
ANDLD
DIFU(013) 302.15  ; 料盒拨料气缸2缩回[Pls]
LD TR0
LD 302.15  ; 料盒拨料气缸2缩回[Pls]
OR 402.15  ; 料盒拨料气缸2缩回[M]
ANDLD
ANDNOT 303.00  ; 料盒拨料气缸2伸出[Pls]
ANDNOT 602.15  ; 料盒拨料气缸2缩回[A]
ANDNOT 603.00  ; 料盒拨料气缸2伸出[A]
ANDNOT 802.15  ; 料盒拨料气缸2原位标志[0002.15]
OUT 402.15  ; 料盒拨料气缸2缩回[M]
LD TR0
AND 703.00  ; 料盒拨料气缸2伸出[SW]
DIFU(013) 303.00  ; 料盒拨料气缸2伸出[Pls]
LD TR0
LD 303.00  ; 料盒拨料气缸2伸出[Pls]
OR 403.00  ; 料盒拨料气缸2伸出[M]
ANDLD
ANDNOT 302.15  ; 料盒拨料气缸2缩回[Pls]
ANDNOT 602.15  ; 料盒拨料气缸2缩回[A]
ANDNOT 603.00  ; 料盒拨料气缸2伸出[A]
ANDNOT 803.00  ; 料盒拨料气缸2到位标志[0003.00]
OUT 403.00  ; 料盒拨料气缸2伸出[M]
; rung 6: 入钉NG收料拉带
LD W1.00  ; 手动模式
ANDNOT D1086.00  ; 入钉NG抓取机构单步/自动循环运行
LD 703.08  ; 入钉NG收料拉带启动[SW]
OR 403.08  ; 入钉NG收料拉带启动[M]
ANDLD
ANDNOT 712.04  ; 入钉NG收料拉带停止[SW]
OUT 403.08  ; 入钉NG收料拉带启动[M]
; rung 7
ILC(003)

### Section 自动程序

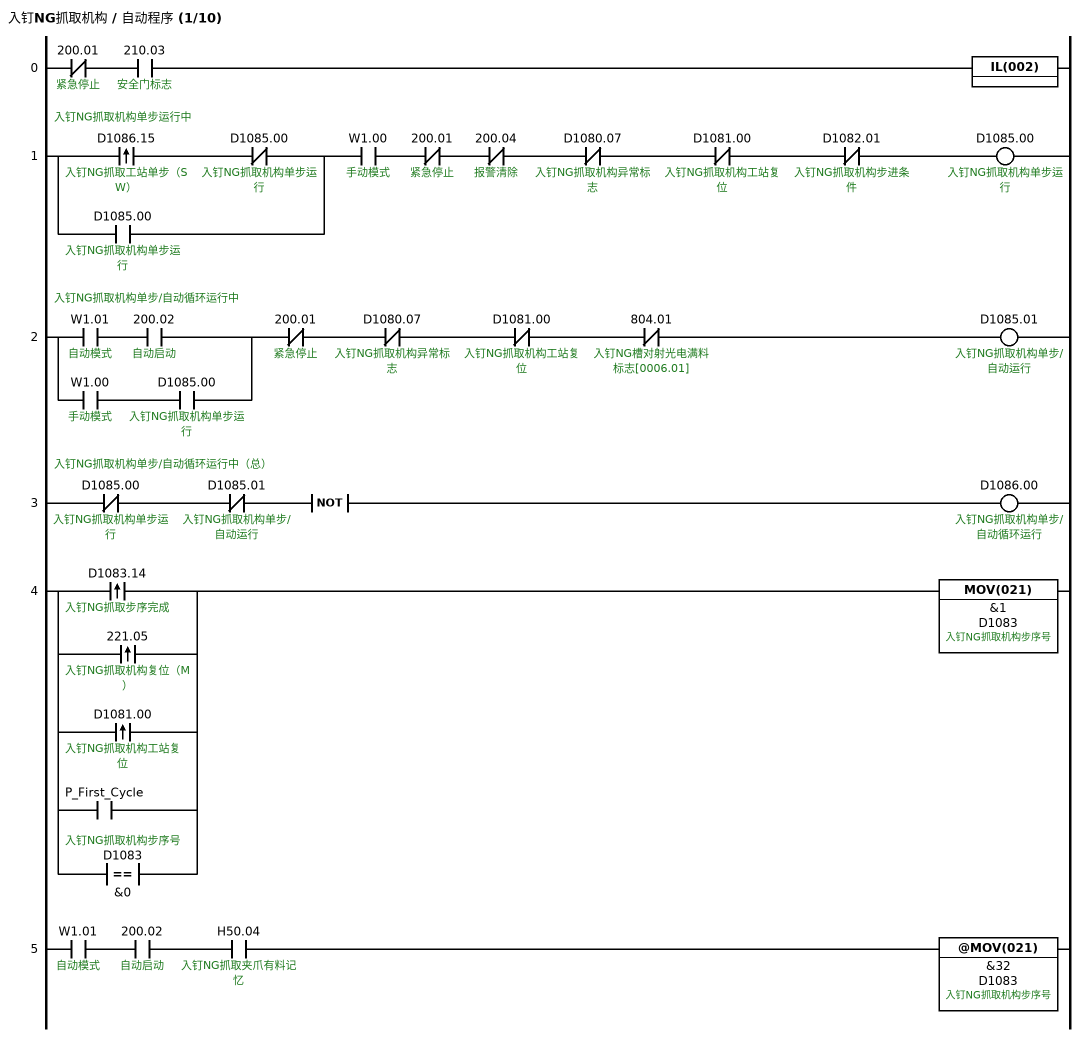
; rung 0
LDNOT 200.01  ; 紧急停止
AND 210.03  ; 安全门标志
IL(002)
; rung 1: 入钉NG抓取机构单步运行中
@LD D1086.15  ; 入钉NG抓取工站单步（SW）
ANDNOT D1085.00  ; 入钉NG抓取机构单步运行
OR D1085.00  ; 入钉NG抓取机构单步运行
AND W1.00  ; 手动模式
ANDNOT 200.01  ; 紧急停止
ANDNOT 200.04  ; 报警清除
ANDNOT D1080.07  ; 入钉NG抓取机构异常标志
ANDNOT D1081.00  ; 入钉NG抓取机构工站复位
ANDNOT D1082.01  ; 入钉NG抓取机构步进条件
OUT D1085.00  ; 入钉NG抓取机构单步运行
; rung 2: 入钉NG抓取机构单步/自动循环运行中
LD W1.01  ; 自动模式
AND 200.02  ; 自动启动
LD W1.00  ; 手动模式
AND D1085.00  ; 入钉NG抓取机构单步运行
ORLD
ANDNOT 200.01  ; 紧急停止
ANDNOT D1080.07  ; 入钉NG抓取机构异常标志
ANDNOT D1081.00  ; 入钉NG抓取机构工站复位
ANDNOT 804.01  ; 入钉NG槽对射光电满料标志[0006.01]
OUT D1085.01  ; 入钉NG抓取机构单步/自动运行
; rung 3: 入钉NG抓取机构单步/自动循环运行中（总）
LDNOT D1085.00  ; 入钉NG抓取机构单步运行
ANDNOT D1085.01  ; 入钉NG抓取机构单步/自动运行
NOT(520)
OUT D1086.00  ; 入钉NG抓取机构单步/自动循环运行
; rung 4
@LD D1083.14  ; 入钉NG抓取步序完成
@OR 221.05  ; 入钉NG抓取机构复位（M）
@OR D1081.00  ; 入钉NG抓取机构工站复位
OR P_First_Cycle
OR=(300) D1083 &0  ; 入钉NG抓取机构步序号
MOV(021) &1 D1083  ; 入钉NG抓取机构步序号
; rung 5
LD W1.01  ; 自动模式
AND 200.02  ; 自动启动
AND H50.04  ; 入钉NG抓取夹爪有料记忆
@MOV(021) &32 D1083  ; 入钉NG抓取机构步序号

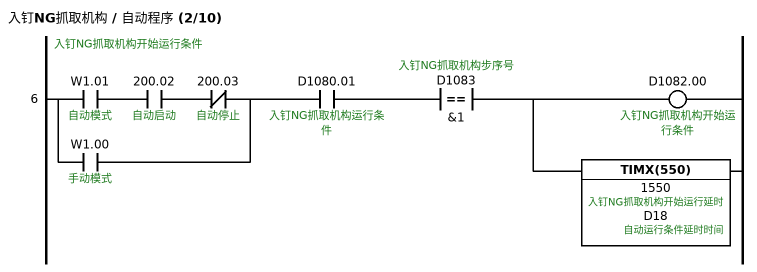
; rung 6: 入钉NG抓取机构开始运行条件
LD W1.01  ; 自动模式
AND 200.02  ; 自动启动
ANDNOT 200.03  ; 自动停止
OR W1.00  ; 手动模式
AND D1080.01  ; 入钉NG抓取机构运行条件
AND=(300) D1083 &1  ; 入钉NG抓取机构步序号
OUT D1082.00  ; 入钉NG抓取机构开始运行条件
TIMX(550) 1550 D18  ; 自动运行条件延时时间, 入钉NG抓取机构开始运行延时

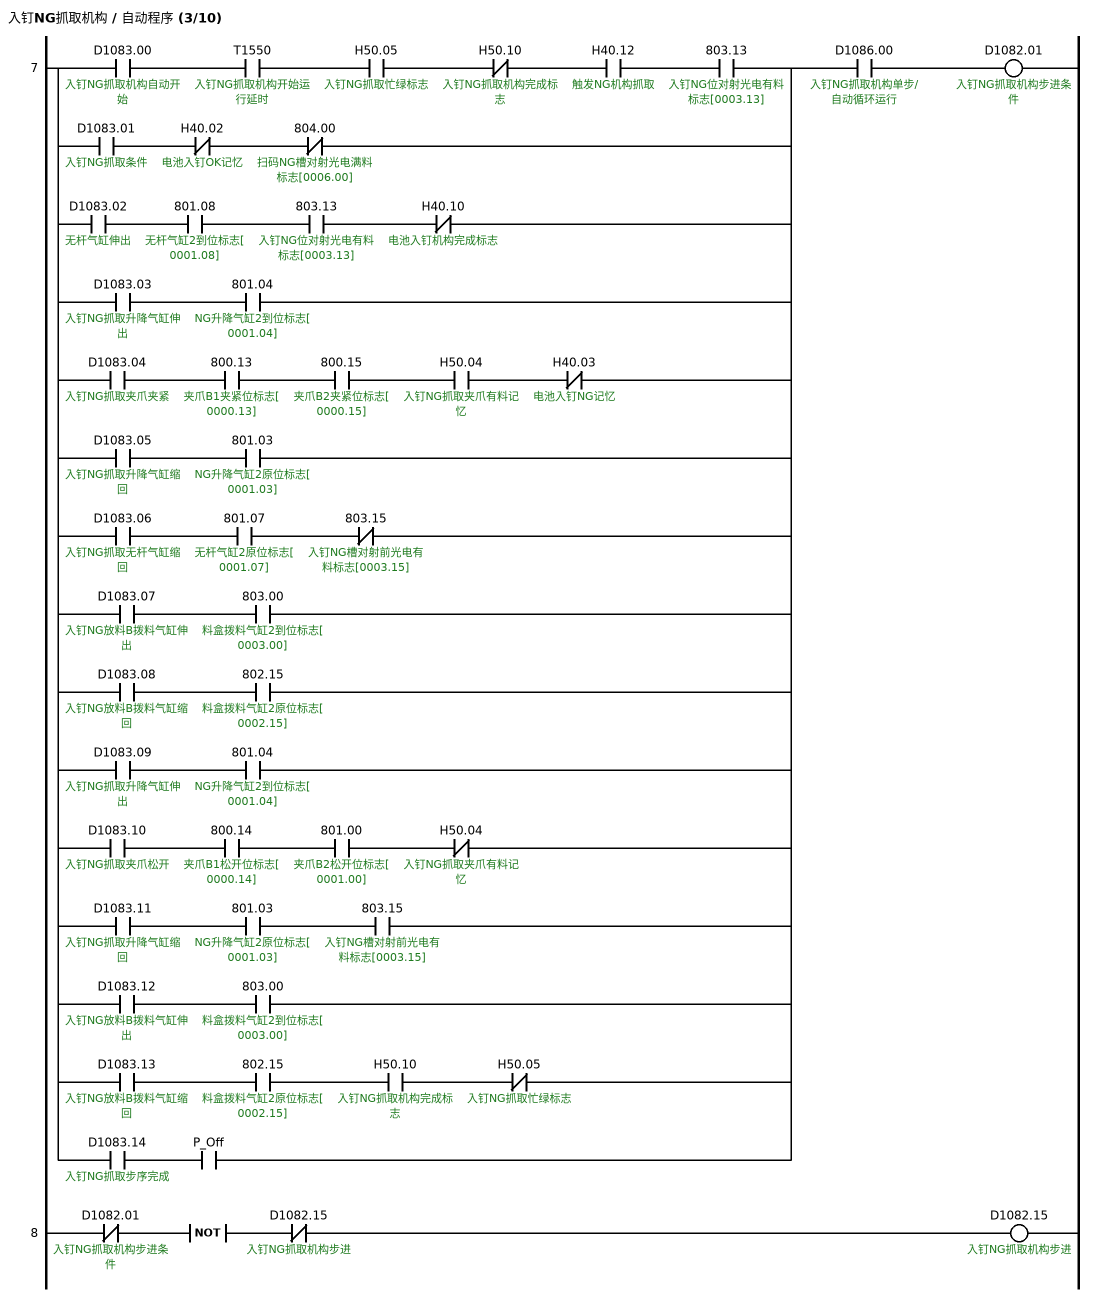
; rung 7
LD D1083.00  ; 入钉NG抓取机构自动开始
AND T1550  ; 入钉NG抓取机构开始运行延时
AND H50.05  ; 入钉NG抓取忙绿标志
ANDNOT H50.10  ; 入钉NG抓取机构完成标志
AND H40.12  ; 触发NG机构抓取
AND 803.13  ; 入钉NG位对射光电有料标志[0003.13]
LD D1083.01  ; 入钉NG抓取条件
ANDNOT H40.02  ; 电池入钉OK记忆
ANDNOT 804.00  ; 扫码NG槽对射光电满料标志[0006.00]
ORLD
LD D1083.02  ; 无杆气缸伸出
AND 801.08  ; 无杆气缸2到位标志[0001.08]
AND 803.13  ; 入钉NG位对射光电有料标志[0003.13]
ANDNOT H40.10  ; 电池入钉机构完成标志
ORLD
LD D1083.03  ; 入钉NG抓取升降气缸伸出
AND 801.04  ; NG升降气缸2到位标志[0001.04]
ORLD
LD D1083.04  ; 入钉NG抓取夹爪夹紧
AND 800.13  ; 夹爪B1夹紧位标志[0000.13]
AND 800.15  ; 夹爪B2夹紧位标志[0000.15]
AND H50.04  ; 入钉NG抓取夹爪有料记忆
ANDNOT H40.03  ; 电池入钉NG记忆
ORLD
LD D1083.05  ; 入钉NG抓取升降气缸缩回
AND 801.03  ; NG升降气缸2原位标志[0001.03]
ORLD
LD D1083.06  ; 入钉NG抓取无杆气缸缩回
AND 801.07  ; 无杆气缸2原位标志[0001.07]
ANDNOT 803.15  ; 入钉NG槽对射前光电有料标志[0003.15]
ORLD
LD D1083.07  ; 入钉NG放料B拨料气缸伸出
AND 803.00  ; 料盒拨料气缸2到位标志[0003.00]
ORLD
LD D1083.08  ; 入钉NG放料B拨料气缸缩回
AND 802.15  ; 料盒拨料气缸2原位标志[0002.15]
ORLD
LD D1083.09  ; 入钉NG抓取升降气缸伸出
AND 801.04  ; NG升降气缸2到位标志[0001.04]
ORLD
LD D1083.10  ; 入钉NG抓取夹爪松开
AND 800.14  ; 夹爪B1松开位标志[0000.14]
AND 801.00  ; 夹爪B2松开位标志[0001.00]
ANDNOT H50.04  ; 入钉NG抓取夹爪有料记忆
ORLD
LD D1083.11  ; 入钉NG抓取升降气缸缩回
AND 801.03  ; NG升降气缸2原位标志[0001.03]
AND 803.15  ; 入钉NG槽对射前光电有料标志[0003.15]
ORLD
LD D1083.12  ; 入钉NG放料B拨料气缸伸出
AND 803.00  ; 料盒拨料气缸2到位标志[0003.00]
ORLD
LD D1083.13  ; 入钉NG放料B拨料气缸缩回
AND 802.15  ; 料盒拨料气缸2原位标志[0002.15]
AND H50.10  ; 入钉NG抓取机构完成标志
ANDNOT H50.05  ; 入钉NG抓取忙绿标志
ORLD
LD D1083.14  ; 入钉NG抓取步序完成
AND P_Off
ORLD
AND D1086.00  ; 入钉NG抓取机构单步/自动循环运行
OUT D1082.01  ; 入钉NG抓取机构步进条件
; rung 8
LDNOT D1082.01  ; 入钉NG抓取机构步进条件
NOT(520)
ANDNOT D1082.15  ; 入钉NG抓取机构步进
OUT D1082.15  ; 入钉NG抓取机构步进

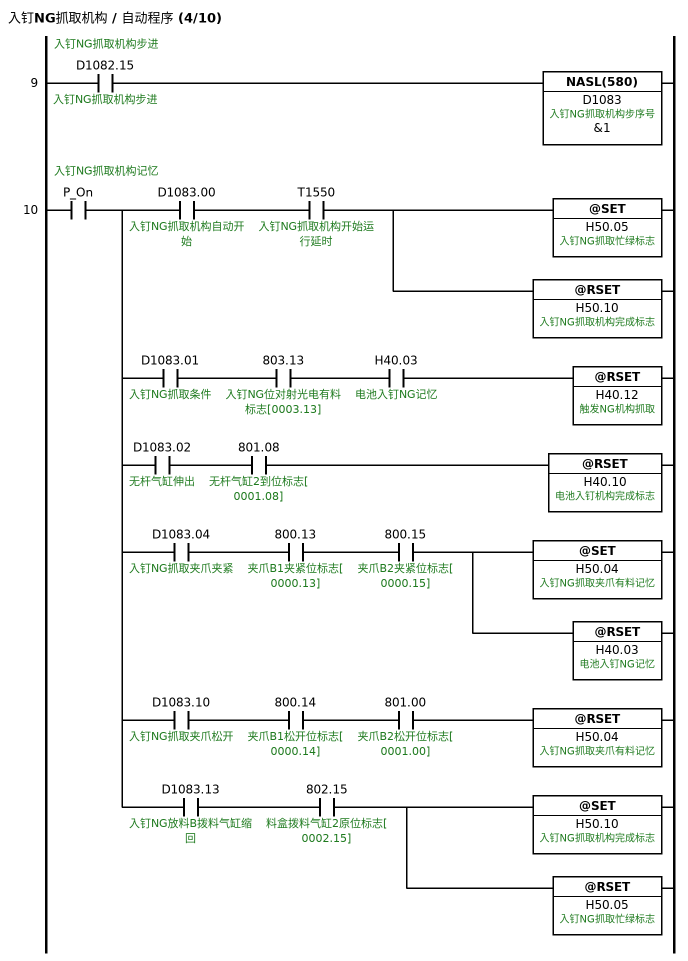
; rung 9: 入钉NG抓取机构步进
LD D1082.15  ; 入钉NG抓取机构步进
NASL(580) D1083 &1  ; 入钉NG抓取机构步序号
; rung 10: 入钉NG抓取机构记忆
LD P_On
OUT TR0
AND D1083.00  ; 入钉NG抓取机构自动开始
AND T1550  ; 入钉NG抓取机构开始运行延时
@SET H50.05  ; 入钉NG抓取忙绿标志
@RSET H50.10  ; 入钉NG抓取机构完成标志
LD TR0
AND D1083.01  ; 入钉NG抓取条件
AND 803.13  ; 入钉NG位对射光电有料标志[0003.13]
AND H40.03  ; 电池入钉NG记忆
@RSET H40.12  ; 触发NG机构抓取
LD TR0
AND D1083.02  ; 无杆气缸伸出
AND 801.08  ; 无杆气缸2到位标志[0001.08]
@RSET H40.10  ; 电池入钉机构完成标志
LD TR0
AND D1083.04  ; 入钉NG抓取夹爪夹紧
AND 800.13  ; 夹爪B1夹紧位标志[0000.13]
AND 800.15  ; 夹爪B2夹紧位标志[0000.15]
@SET H50.04  ; 入钉NG抓取夹爪有料记忆
@RSET H40.03  ; 电池入钉NG记忆
LD TR0
AND D1083.10  ; 入钉NG抓取夹爪松开
AND 800.14  ; 夹爪B1松开位标志[0000.14]
AND 801.00  ; 夹爪B2松开位标志[0001.00]
@RSET H50.04  ; 入钉NG抓取夹爪有料记忆
LD TR0
AND D1083.13  ; 入钉NG放料B拨料气缸缩回
AND 802.15  ; 料盒拨料气缸2原位标志[0002.15]
@SET H50.10  ; 入钉NG抓取机构完成标志
@RSET H50.05  ; 入钉NG抓取忙绿标志

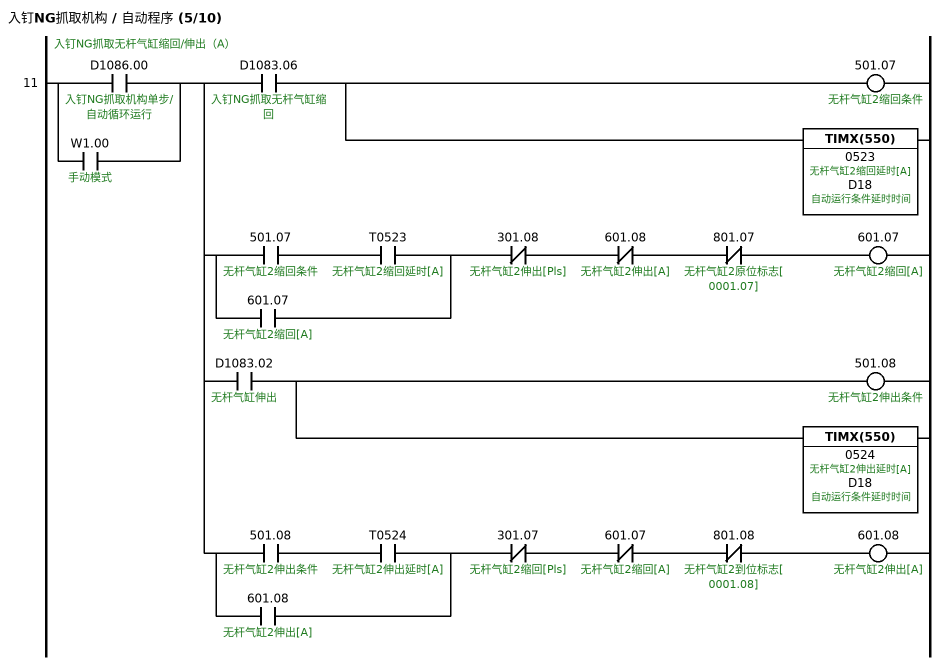
; rung 11: 入钉NG抓取无杆气缸缩回/伸出（A）
LD D1086.00  ; 入钉NG抓取机构单步/自动循环运行
OR W1.00  ; 手动模式
OUT TR0
AND D1083.06  ; 入钉NG抓取无杆气缸缩回
OUT 501.07  ; 无杆气缸2缩回条件
TIMX(550) 0523 D18  ; 自动运行条件延时时间, 无杆气缸2缩回延时[A]
LD TR0
LD 501.07  ; 无杆气缸2缩回条件
AND T0523  ; 无杆气缸2缩回延时[A]
OR 601.07  ; 无杆气缸2缩回[A]
ANDLD
ANDNOT 301.08  ; 无杆气缸2伸出[Pls]
ANDNOT 601.08  ; 无杆气缸2伸出[A]
ANDNOT 801.07  ; 无杆气缸2原位标志[0001.07]
OUT 601.07  ; 无杆气缸2缩回[A]
LD TR0
AND D1083.02  ; 无杆气缸伸出
OUT 501.08  ; 无杆气缸2伸出条件
TIMX(550) 0524 D18  ; 自动运行条件延时时间, 无杆气缸2伸出延时[A]
LD TR0
LD 501.08  ; 无杆气缸2伸出条件
AND T0524  ; 无杆气缸2伸出延时[A]
OR 601.08  ; 无杆气缸2伸出[A]
ANDLD
ANDNOT 301.07  ; 无杆气缸2缩回[Pls]
ANDNOT 601.07  ; 无杆气缸2缩回[A]
ANDNOT 801.08  ; 无杆气缸2到位标志[0001.08]
OUT 601.08  ; 无杆气缸2伸出[A]

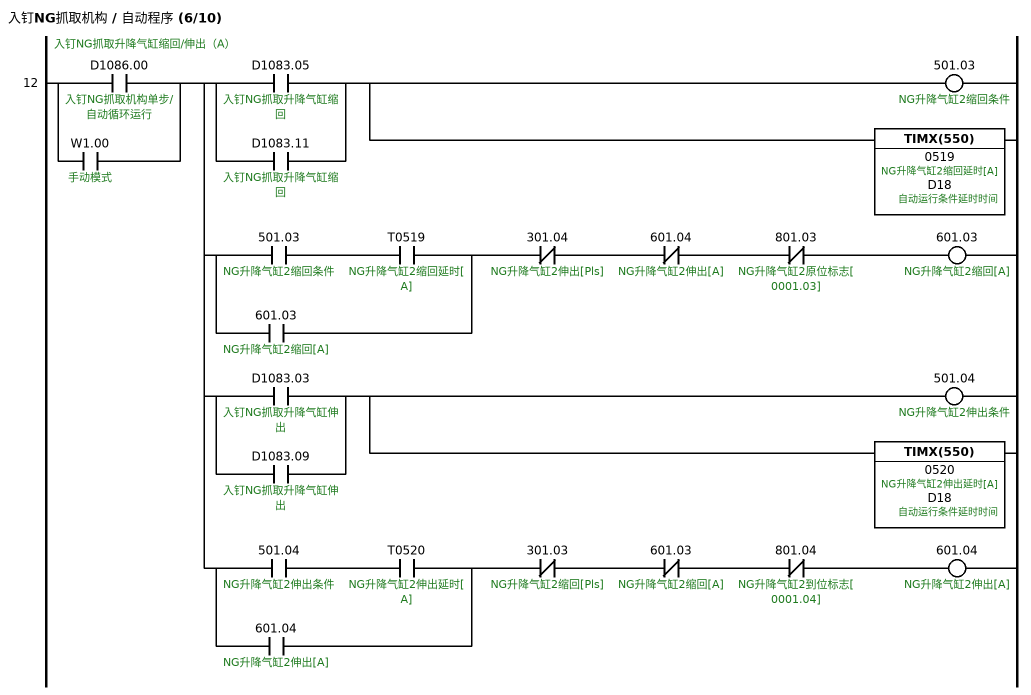
; rung 12: 入钉NG抓取升降气缸缩回/伸出（A）
LD D1086.00  ; 入钉NG抓取机构单步/自动循环运行
OR W1.00  ; 手动模式
OUT TR0
LD D1083.05  ; 入钉NG抓取升降气缸缩回
OR D1083.11  ; 入钉NG抓取升降气缸缩回
ANDLD
OUT 501.03  ; NG升降气缸2缩回条件
TIMX(550) 0519 D18  ; 自动运行条件延时时间, NG升降气缸2缩回延时[A]
LD TR0
LD 501.03  ; NG升降气缸2缩回条件
AND T0519  ; NG升降气缸2缩回延时[A]
OR 601.03  ; NG升降气缸2缩回[A]
ANDLD
ANDNOT 301.04  ; NG升降气缸2伸出[Pls]
ANDNOT 601.04  ; NG升降气缸2伸出[A]
ANDNOT 801.03  ; NG升降气缸2原位标志[0001.03]
OUT 601.03  ; NG升降气缸2缩回[A]
LD TR0
LD D1083.03  ; 入钉NG抓取升降气缸伸出
OR D1083.09  ; 入钉NG抓取升降气缸伸出
ANDLD
OUT 501.04  ; NG升降气缸2伸出条件
TIMX(550) 0520 D18  ; 自动运行条件延时时间, NG升降气缸2伸出延时[A]
LD TR0
LD 501.04  ; NG升降气缸2伸出条件
AND T0520  ; NG升降气缸2伸出延时[A]
OR 601.04  ; NG升降气缸2伸出[A]
ANDLD
ANDNOT 301.03  ; NG升降气缸2缩回[Pls]
ANDNOT 601.03  ; NG升降气缸2缩回[A]
ANDNOT 801.04  ; NG升降气缸2到位标志[0001.04]
OUT 601.04  ; NG升降气缸2伸出[A]

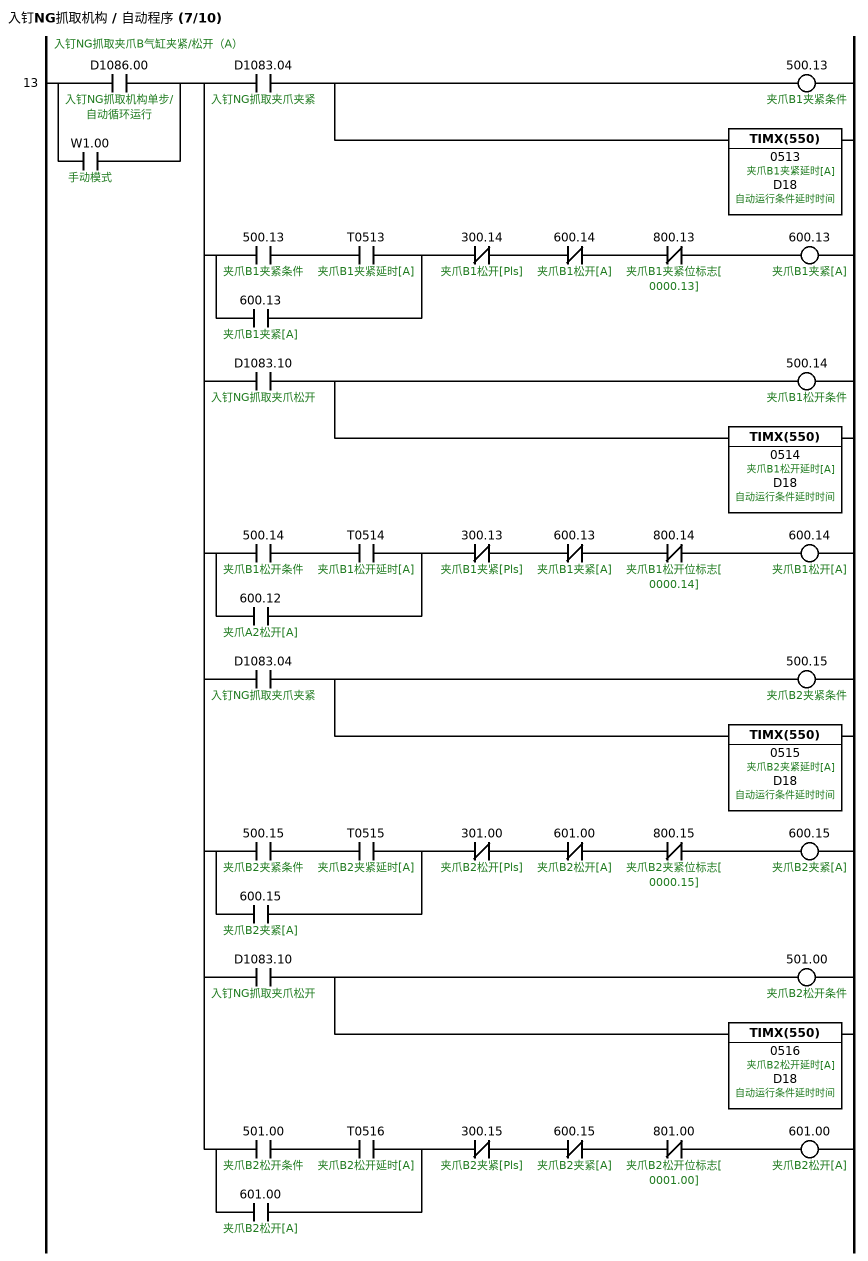
; rung 13: 入钉NG抓取夹爪B气缸夹紧/松开（A）
LD D1086.00  ; 入钉NG抓取机构单步/自动循环运行
OR W1.00  ; 手动模式
OUT TR0
AND D1083.04  ; 入钉NG抓取夹爪夹紧
OUT 500.13  ; 夹爪B1夹紧条件
TIMX(550) 0513 D18  ; 自动运行条件延时时间, 夹爪B1夹紧延时[A]
LD TR0
LD 500.13  ; 夹爪B1夹紧条件
AND T0513  ; 夹爪B1夹紧延时[A]
OR 600.13  ; 夹爪B1夹紧[A]
ANDLD
ANDNOT 300.14  ; 夹爪B1松开[Pls]
ANDNOT 600.14  ; 夹爪B1松开[A]
ANDNOT 800.13  ; 夹爪B1夹紧位标志[0000.13]
OUT 600.13  ; 夹爪B1夹紧[A]
LD TR0
AND D1083.10  ; 入钉NG抓取夹爪松开
OUT 500.14  ; 夹爪B1松开条件
TIMX(550) 0514 D18  ; 自动运行条件延时时间, 夹爪B1松开延时[A]
LD TR0
LD 500.14  ; 夹爪B1松开条件
AND T0514  ; 夹爪B1松开延时[A]
OR 600.12  ; 夹爪A2松开[A]
ANDLD
ANDNOT 300.13  ; 夹爪B1夹紧[Pls]
ANDNOT 600.13  ; 夹爪B1夹紧[A]
ANDNOT 800.14  ; 夹爪B1松开位标志[0000.14]
OUT 600.14  ; 夹爪B1松开[A]
LD TR0
AND D1083.04  ; 入钉NG抓取夹爪夹紧
OUT 500.15  ; 夹爪B2夹紧条件
TIMX(550) 0515 D18  ; 自动运行条件延时时间, 夹爪B2夹紧延时[A]
LD TR0
LD 500.15  ; 夹爪B2夹紧条件
AND T0515  ; 夹爪B2夹紧延时[A]
OR 600.15  ; 夹爪B2夹紧[A]
ANDLD
ANDNOT 301.00  ; 夹爪B2松开[Pls]
ANDNOT 601.00  ; 夹爪B2松开[A]
ANDNOT 800.15  ; 夹爪B2夹紧位标志[0000.15]
OUT 600.15  ; 夹爪B2夹紧[A]
LD TR0
AND D1083.10  ; 入钉NG抓取夹爪松开
OUT 501.00  ; 夹爪B2松开条件
TIMX(550) 0516 D18  ; 自动运行条件延时时间, 夹爪B2松开延时[A]
LD TR0
LD 501.00  ; 夹爪B2松开条件
AND T0516  ; 夹爪B2松开延时[A]
OR 601.00  ; 夹爪B2松开[A]
ANDLD
ANDNOT 300.15  ; 夹爪B2夹紧[Pls]
ANDNOT 600.15  ; 夹爪B2夹紧[A]
ANDNOT 801.00  ; 夹爪B2松开位标志[0001.00]
OUT 601.00  ; 夹爪B2松开[A]

